PROGRAM MAIN
VAR	
END_VAR

VAR_INPUT
	qxABBonlineLamp : BOOL;
	qxABBExecutLamp : BOOL;
	qxABBErrorLamp : BOOL;
	qxPauseLamp : BOOL;
	qxEmergySTLamp : BOOL;
	ixPauseButt : BOOL;
	ixResetABB : BOOL;
	qxAutoMode : BOOL;
	qxManualMode : BOOL;
	ixAutoLamp : BOOL;
	ixManualLamp : BOOL;
	qxDoneContainerScan : BOOL;
	qxDoneBuffer1Scan : BOOL;
	qsContainer : STRING;
	qsTask : STRING;
	qsSubTask : STRING;
	mxPlateAvailable : BOOL;
	mxCylinderAvailable : BOOL;
	mxOctagonAvailable : BOOL;
	mwBufferID : INT;
	ixEmptyBuffer : BOOL;
	mwPartID : INT;
	sPartID : ARRAY [1..3] OF STRING:= ['Part 1', 'Part 2', 'Part 3'];
END_VAR

VAR_OUTPUT
	
END_VAR

AutomationLibrary();
Visualaisation_Control();
RobotPosTracker();
ABB_Control_FB();

END_PROGRAM

(* stored: Version 1.1.0.1, ProductVersion 3.1.4024.12
   POU MAIN: Id {eedc87b0-498f-42a3-9add-b62d0d4a527c}, SpecialFunc None *)
